// TIA Portal V20 export
// export: Created 2025-12-01T14:57:14.6976508Z, ExportSetting None, DisplayName Totally Integrated Automation Portal, DisplayVersion V20 Update 3, DisplayName TIA Portal Openness, DisplayVersion V20 Update 3, DisplayName TIA Portal Version Control Interface, DisplayVersion V20 Update 3, DisplayName STEP 7 Professional, DisplayVersion V20 Update 3, DisplayName STEP 7 Safety, DisplayVersion V20 Update 2, DisplayName WinCC Basic/Comfort/Advanced, DisplayVersion V20 Update 3, DisplayName WinCC Professional, DisplayVersion V20 Update 3, DisplayName WinCC Unified, DisplayVersion V20 Update 3
FUNCTION "FC901_Marcas_Auxiliares" : Void   // FC901, LAD
{ S7_Optimized_Access := 'FALSE' }
AUTHOR : GENERAL
NAME : 20130301
VERSION : 3.0
// stored: AutoNumber false, SetENOAutomatically false
   VAR_TEMP
      Incremento_Tiempo : Time;
      Aux_Ret_Val : Int;
      Fecha_Actual : Date;
      Hora : Time_Of_Day;
      Fecha_y_hora : Date_And_Time;
      troceado AT Fecha_y_hora : Struct
         año : Byte;
         mes : Byte;
         dia : Byte;
         hora : Byte;
         minuto : Byte;
         segundo : Byte;
         ms : Byte;
         "ms2+d_sem" : Byte;
      END_STRUCT;
      retval : Int;
      hora_convertida : ULInt;
      hora_total_string : String[9];
      hora_int : ULInt;
      minuto_int : ULInt;
      segundo_int : ULInt;
      milisegundo_int : ULInt;
   END_VAR
   VAR_TEMP   // added for the SCL form of the ladder/FBD networks
      _w1 : Bool;
   END_VAR
BEGIN

REGION Network 1: Marca que siempre esta a ON
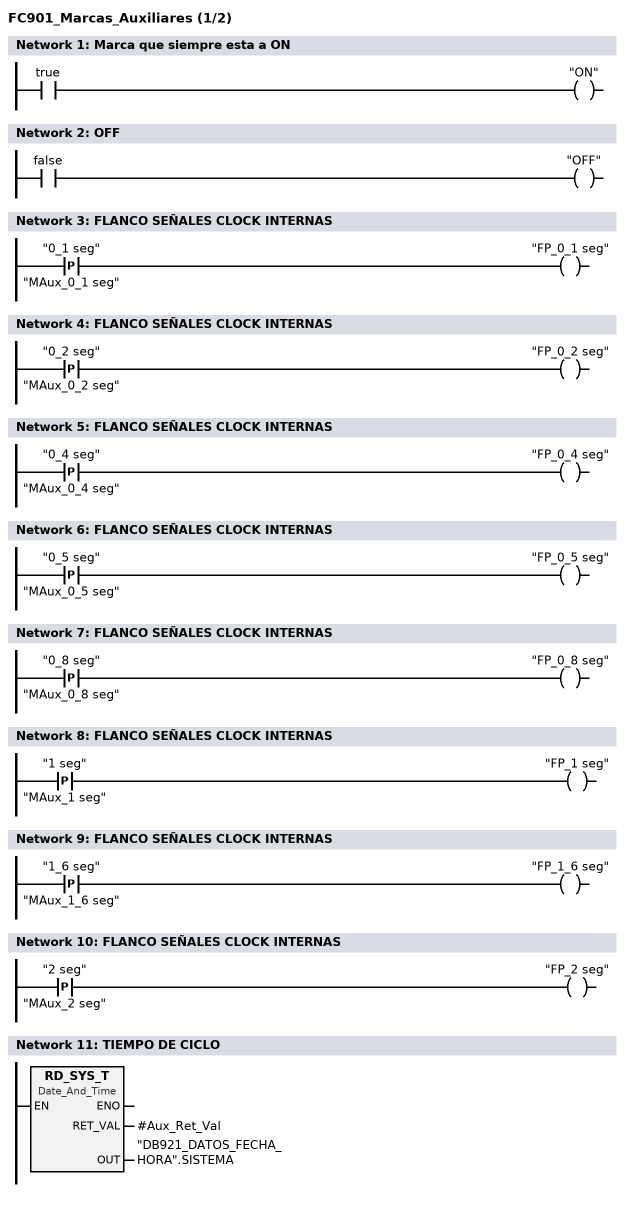
   RUNG wire#powerrail
      Contact( true )
      Coil( "ON" )
   END_RUNG
   // the same network as SCL:
   "ON" := true;
END_REGION

REGION Network 2: OFF
   RUNG wire#powerrail
      Contact( false )
      Coil( "OFF" )
   END_RUNG
   // the same network as SCL:
   "OFF" := false;
END_REGION

REGION Network 3: FLANCO SEÑALES CLOCK INTERNAS
   RUNG wire#powerrail
      P_Contact(operand := "0_1 seg", bit := "MAux_0_1 seg")
      Coil( "FP_0_1 seg" )
   END_RUNG
   // the same network as SCL:
   #_w1 := "0_1 seg" AND NOT "MAux_0_1 seg";   // rising edge of "0_1 seg"
   "MAux_0_1 seg" := "0_1 seg";
   "FP_0_1 seg" := #_w1;
END_REGION

REGION Network 4: FLANCO SEÑALES CLOCK INTERNAS
   RUNG wire#powerrail
      P_Contact(operand := "0_2 seg", bit := "MAux_0_2 seg")
      Coil( "FP_0_2 seg" )
   END_RUNG
   // the same network as SCL:
   #_w1 := "0_2 seg" AND NOT "MAux_0_2 seg";   // rising edge of "0_2 seg"
   "MAux_0_2 seg" := "0_2 seg";
   "FP_0_2 seg" := #_w1;
END_REGION

REGION Network 5: FLANCO SEÑALES CLOCK INTERNAS
   RUNG wire#powerrail
      P_Contact(operand := "0_4 seg", bit := "MAux_0_4 seg")
      Coil( "FP_0_4 seg" )
   END_RUNG
   // the same network as SCL:
   #_w1 := "0_4 seg" AND NOT "MAux_0_4 seg";   // rising edge of "0_4 seg"
   "MAux_0_4 seg" := "0_4 seg";
   "FP_0_4 seg" := #_w1;
END_REGION

REGION Network 6: FLANCO SEÑALES CLOCK INTERNAS
   RUNG wire#powerrail
      P_Contact(operand := "0_5 seg", bit := "MAux_0_5 seg")
      Coil( "FP_0_5 seg" )
   END_RUNG
   // the same network as SCL:
   #_w1 := "0_5 seg" AND NOT "MAux_0_5 seg";   // rising edge of "0_5 seg"
   "MAux_0_5 seg" := "0_5 seg";
   "FP_0_5 seg" := #_w1;
END_REGION

REGION Network 7: FLANCO SEÑALES CLOCK INTERNAS
   RUNG wire#powerrail
      P_Contact(operand := "0_8 seg", bit := "MAux_0_8 seg")
      Coil( "FP_0_8 seg" )
   END_RUNG
   // the same network as SCL:
   #_w1 := "0_8 seg" AND NOT "MAux_0_8 seg";   // rising edge of "0_8 seg"
   "MAux_0_8 seg" := "0_8 seg";
   "FP_0_8 seg" := #_w1;
END_REGION

REGION Network 8: FLANCO SEÑALES CLOCK INTERNAS
   RUNG wire#powerrail
      P_Contact(operand := "1 seg", bit := "MAux_1 seg")
      Coil( "FP_1 seg" )
   END_RUNG
   // the same network as SCL:
   #_w1 := "1 seg" AND NOT "MAux_1 seg";   // rising edge of "1 seg"
   "MAux_1 seg" := "1 seg";
   "FP_1 seg" := #_w1;
END_REGION

REGION Network 9: FLANCO SEÑALES CLOCK INTERNAS
   RUNG wire#powerrail
      P_Contact(operand := "1_6 seg", bit := "MAux_1_6 seg")
      Coil( "FP_1_6 seg" )
   END_RUNG
   // the same network as SCL:
   #_w1 := "1_6 seg" AND NOT "MAux_1_6 seg";   // rising edge of "1_6 seg"
   "MAux_1_6 seg" := "1_6 seg";
   "FP_1_6 seg" := #_w1;
END_REGION

REGION Network 10: FLANCO SEÑALES CLOCK INTERNAS
   RUNG wire#powerrail
      P_Contact(operand := "2 seg", bit := "MAux_2 seg")
      Coil( "FP_2 seg" )
   END_RUNG
   // the same network as SCL:
   #_w1 := "2 seg" AND NOT "MAux_2 seg";   // rising edge of "2 seg"
   "MAux_2 seg" := "2 seg";
   "FP_2 seg" := #_w1;
END_REGION

REGION Network 11: TIEMPO DE CICLO
   RUNG wire#powerrail
      { S7_Templates := "date_type := Date_And_Time" } RD_SYS_T(RET_VAL => #Aux_Ret_Val, OUT => "DB921_DATOS_FECHA_HORA".SISTEMA)
   END_RUNG
   // the same network as SCL:
   #Aux_Ret_Val := RD_SYS_T(OUT => "DB921_DATOS_FECHA_HORA".SISTEMA);
END_REGION

REGION Network 12
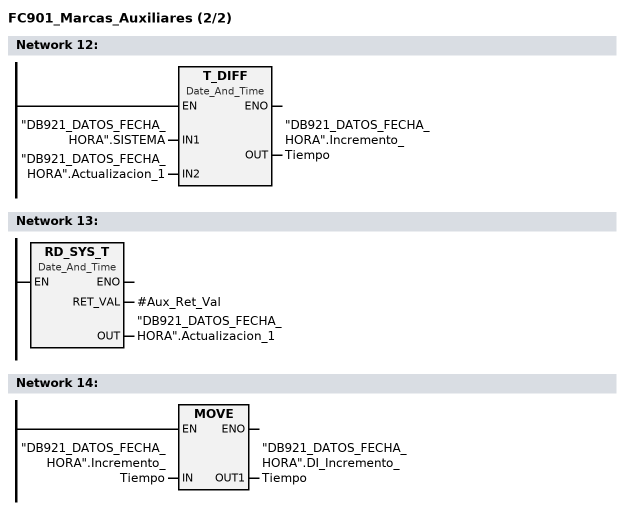
   RUNG wire#powerrail
      { S7_Templates := "[date_type := Date_And_Time, time_type := Time]" } T_DIFF(IN1 := "DB921_DATOS_FECHA_HORA".SISTEMA, IN2 := "DB921_DATOS_FECHA_HORA".Actualizacion_1, OUT => "DB921_DATOS_FECHA_HORA".Incremento_Tiempo)
   END_RUNG
   // the same network as SCL:
   T_DIFF(IN1 := "DB921_DATOS_FECHA_HORA".SISTEMA,
          IN2 := "DB921_DATOS_FECHA_HORA".Actualizacion_1,
          OUT => "DB921_DATOS_FECHA_HORA".Incremento_Tiempo);
END_REGION

REGION Network 13
   RUNG wire#powerrail
      { S7_Templates := "date_type := Date_And_Time" } RD_SYS_T(RET_VAL => #Aux_Ret_Val, OUT => "DB921_DATOS_FECHA_HORA".Actualizacion_1)
   END_RUNG
   // the same network as SCL:
   #Aux_Ret_Val := RD_SYS_T(OUT => "DB921_DATOS_FECHA_HORA".Actualizacion_1);
END_REGION

REGION Network 14
   RUNG wire#powerrail
      { S7_GenerateENO := "TRUE" } Move(in := "DB921_DATOS_FECHA_HORA".Incremento_Tiempo, out1 => "DB921_DATOS_FECHA_HORA".DI_Incremento_Tiempo)
   END_RUNG
   // the same network as SCL:
   "DB921_DATOS_FECHA_HORA".DI_Incremento_Tiempo := "DB921_DATOS_FECHA_HORA".Incremento_Tiempo;
END_REGION

REGION Network 15 (SCL)
   // GENERAR EL SELLO DE TIEMPO PARA LOS MENSAJES
   // 
   IF  "con_sello_tiempo" = true THEN

       REGION formatear_hora

           #retval := RD_LOC_T(#Fecha_y_hora);
           #hora_int := BCD16_TO_INT(#troceado.hora);
           #minuto_int := BCD16_TO_INT(#troceado.minuto);
           #segundo_int := BCD16_TO_INT(#troceado.segundo);
           #milisegundo_int := BCD16_TO_INT(#troceado.ms);
           #hora_convertida := 0;

           #hora_convertida := (#hora_int * 10000000) + (#minuto_int * 100000) + (#segundo_int * 1000) + #milisegundo_int;
           #hora_total_string := DELETE(IN := (ULINT_TO_STRING(IN := #hora_convertida)), L := 1, P := 1);

           "DB921_DATOS_FECHA_HORA".TIME_STAMP := CONCAT(IN1 := '[TIME]', IN2 := #hora_total_string);

       END_REGION

   ELSE
       "DB921_DATOS_FECHA_HORA".TIME_STAMP := '';
   END_IF;
END_REGION
END_FUNCTION
